(* PLC project Verven 4.project, CODESYS CODESYS V3.5 SP19 Patch 7 *)
(* stored: creationDateTime 2024-11-20T06:37:52.120257, modificationDateTime 2024-11-19T14:23:32.9936829 *)

VAR_GLOBAL  (* GVL_ClimateControl *)
  typClimateControllerInterfaceRoomA401_1 : typMultiModeClimateControl_00_01;
  typClimateControllerInterfaceRoomA401_2 : typMultiModeClimateControl_00_01;
  typClimateControllerInterfaceRoomA401_3 : typMultiModeClimateControl_00_01;
  typClimateControllerInterfaceRoomA401_4 : typMultiModeClimateControl_00_01;
  typClimateControllerInterfaceRoomA402 : typMultiModeClimateControl_00_01;
  typClimateControllerInterfaceRoomA403 : typMultiModeClimateControl_00_01;
  typClimateControllerInterfaceRoomA406 : typMultiModeClimateControl_00_01;
  typClimateControllerInterfaceRoomA407 : typMultiModeClimateControl_00_01;
  typClimateControllerInterfaceRoomA408 : typMultiModeClimateControl_00_01;
  typClimateControllerInterfaceRoomA409 : typMultiModeClimateControl_00_01;
  typClimateControllerInterfaceRoomA410_1 : typMultiModeClimateControl_00_01;
  typClimateControllerInterfaceRoomA410_2 : typMultiModeClimateControl_00_01;
  typClimateControllerInterfaceRoomA412 : typMultiModeClimateControl_00_01;
  typClimateControllerInterfaceRoomA413 : typMultiModeClimateControl_00_01;
  typClimateControllerInterfaceRoomA415 : typMultiModeClimateControl_00_01;
  typClimateControllerInterfaceRoomA416 : typMultiModeClimateControl_00_01;
  typClimateControllerInterfaceRoomA417 : typMultiModeClimateControl_00_01;
  typClimateControllerInterfaceRoomA418 : typMultiModeClimateControl_00_01;
  typClimateControllerInterfaceRoomA425 : typMultiModeClimateControl_00_01;
  typClimateControllerInterfaceRoomA426 : typMultiModeClimateControl_00_01;
  typClimateControllerInterfaceRoomA427 : typMultiModeClimateControl_00_01;
  typClimateControllerInterfaceRoomA428 : typMultiModeClimateControl_00_01;
  typClimateControllerInterfaceRoomA428_1 : typMultiModeClimateControl_00_01;
  typClimateControllerInterfaceRoomA428_2 : typMultiModeClimateControl_00_01;
  typClimateControllerInterfaceRoomA428_3 : typMultiModeClimateControl_00_01;
  typClimateControllerInterfaceRoomA430 : typMultiModeClimateControl_00_01;
END_VAR
